// TIA Portal V20 export
DATA_BLOCK "AlarmWords"   // DB93
   VAR
      AlarmWord1 : Word;
      AlarmWord0 : Word;
      AlarmWord2 : Word;
      AlarmWord3 : Word;
   END_VAR
BEGIN
END_DATA_BLOCK
